SUBAPPLICATION mapping (* Subapplication Type *)
  (* Standard: 61499-2 *)
  (* Version 1.0, 2023-10-23, franz *)
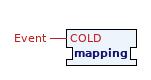
  EVENT_INPUT
    COLD;
  END_EVENT
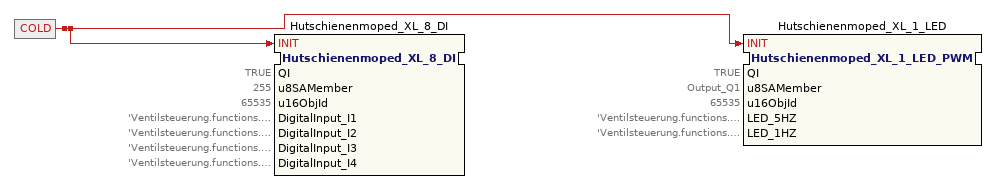
  (* BUTTON_PRESS_NORMAL *)
  FBS
    Hutschienenmoped_XL_8_DI : Hutschienenmoped_XL_8_DI(QI := TRUE, u8SAMember := 255, u16ObjId := 65535, DigitalInput_I1 := 'Ventilsteuerung.functions.DigitalInput_I1', DigitalInput_I2 := 'Ventilsteuerung.functions.DigitalInput_I2', DigitalInput_I3 := 'Ventilsteuerung.functions.DigitalInput_I3', DigitalInput_I4 := 'Ventilsteuerung.functions.DigitalInput_I4');
    Hutschienenmoped_XL_1_LED : Hutschienenmoped_XL_1_LED_PWM(QI := TRUE, u8SAMember := Output_Q1, u16ObjId := 65535, LED_5HZ := 'Ventilsteuerung.functions.LED_Q1_5HZ', LED_1HZ := 'Ventilsteuerung.functions.LED_Q1_1HZ');
  END_FBS
  EVENT_CONNECTIONS
    COLD TO Hutschienenmoped_XL_8_DI.INIT;
    COLD TO Hutschienenmoped_XL_1_LED.INIT;
  END_CONNECTIONS
END_SUBAPPLICATION
